FUNCTION_BLOCK SM_BaseMcProcess EXTENDS BaseProcess
VAR_INPUT
	///Error ID according to Beckhoff/PlcOpen Motion Control
	{attribute 'OPC.UA.DA' := '1'}
	{attribute 'OPC.UA.DA.Access' := '1'}
	errorId: UDINT;
END_VAR
VAR_OUTPUT
END_VAR
VAR_IN_OUT
END_VAR
VAR
END_VAR

SUPER^();

END_FUNCTION_BLOCK

(* stored: Version 1.1.0.1, ProductVersion 3.1.4019.2
   POU SM_BaseMcProcess: Id {48332927-2c6f-40f2-b025-117b81e810d4}, SpecialFunc None *)
